// Mitsubishi GX Works2 project: 모터제어   PLC: Q03UDV

PROGRAM MAIN
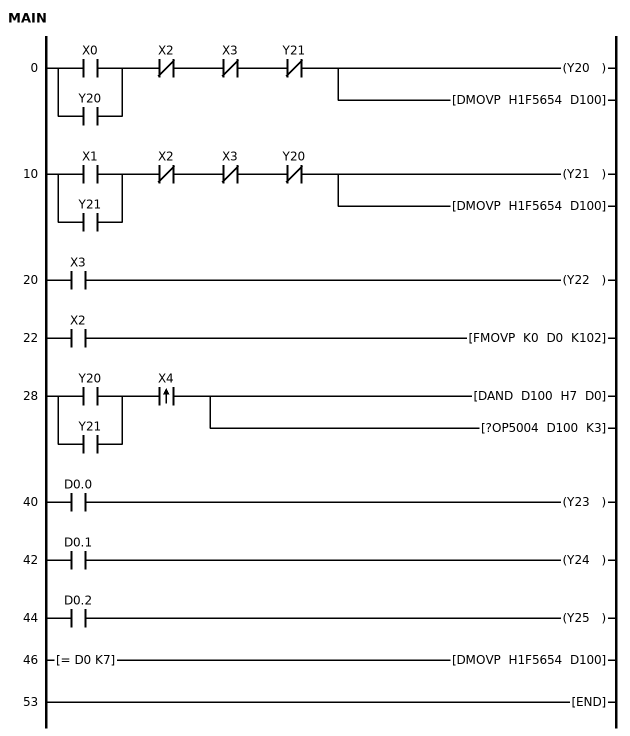
0     LD      X0
      OR      Y20
      ANI     X2
      ANI     X3
      ANI     Y21
      OUT     Y20
      DMOVP   H1F5654 D100
10    LD      X1
      OR      Y21
      ANI     X2
      ANI     X3
      ANI     Y20
      OUT     Y21
      DMOVP   H1F5654 D100
20    LD      X3
      OUT     Y22
22    LD      X2
      FMOVP   K0 D0 K102
28    LD      Y20
      OR      Y21
      ANDP    X4
      DAND    D100 H7 D0
      ?OP5004 D100 K3
40    LD      D0.0
      OUT     Y23
42    LD      D0.1
      OUT     Y24
44    LD      D0.2
      OUT     Y25
46    LD=     D0 K7
      DMOVP   H1F5654 D100
53    END
END_PROGRAM
